FUNCTION_BLOCK jobServiceInterface (* Composite Function Block Type *)
  (* Standard: 61499-2 *)
  (* Version 0.0, 2018-03-05, 4DIAC-IDE, 4DIAC-Consortium *)
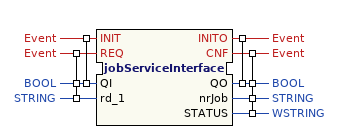
  EVENT_INPUT
    INIT WITH QI; (* Initialization Request *)
    REQ WITH QI, rd_1; (* Normal Execution Request *)
  END_EVENT
  EVENT_OUTPUT
    INITO WITH QO; (* Initialization Confirm *)
    CNF WITH QO, nrJob, STATUS; (* Execution Confirmation *)
  END_EVENT
  VAR_INPUT
    QI : BOOL := TRUE; (* Input event qualifier *)
    rd_1 : STRING;
  END_VAR
  VAR_OUTPUT
    QO : BOOL; (* Output event qualifier *)
    nrJob : STRING;
    STATUS : WSTRING;
  END_VAR
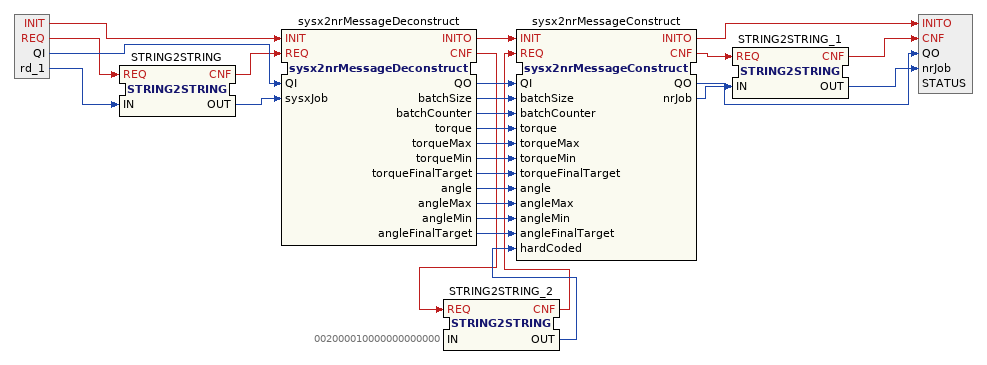
  FBS
    STRING2STRING : STRING2STRING;
    sysx2nrMessageDeconstruct : sysx2nrMessageDeconstruct;
    sysx2nrMessageConstruct : sysx2nrMessageConstruct;
    STRING2STRING_1 : STRING2STRING;
    STRING2STRING_2 : STRING2STRING(IN := 002000010000000000000);
  END_FBS
  EVENT_CONNECTIONS
    STRING2STRING.CNF TO sysx2nrMessageDeconstruct.REQ;
    sysx2nrMessageDeconstruct.INITO TO sysx2nrMessageConstruct.INIT;
    sysx2nrMessageConstruct.INITO TO INITO;
    STRING2STRING_1.CNF TO CNF;
    sysx2nrMessageConstruct.CNF TO STRING2STRING_1.REQ;
    REQ TO STRING2STRING.REQ;
    INIT TO sysx2nrMessageDeconstruct.INIT;
    sysx2nrMessageDeconstruct.CNF TO STRING2STRING_2.REQ;
    STRING2STRING_2.CNF TO sysx2nrMessageConstruct.REQ;
  END_CONNECTIONS
  DATA_CONNECTIONS
    STRING2STRING.OUT TO sysx2nrMessageDeconstruct.sysxJob;
    sysx2nrMessageDeconstruct.QO TO sysx2nrMessageConstruct.QI;
    sysx2nrMessageDeconstruct.batchSize TO sysx2nrMessageConstruct.batchSize;
    sysx2nrMessageDeconstruct.batchCounter TO sysx2nrMessageConstruct.batchCounter;
    sysx2nrMessageDeconstruct.torque TO sysx2nrMessageConstruct.torque;
    sysx2nrMessageDeconstruct.torqueMax TO sysx2nrMessageConstruct.torqueMax;
    sysx2nrMessageDeconstruct.torqueMin TO sysx2nrMessageConstruct.torqueMin;
    sysx2nrMessageDeconstruct.torqueFinalTarget TO sysx2nrMessageConstruct.torqueFinalTarget;
    sysx2nrMessageDeconstruct.angle TO sysx2nrMessageConstruct.angle;
    sysx2nrMessageDeconstruct.angleMax TO sysx2nrMessageConstruct.angleMax;
    sysx2nrMessageDeconstruct.angleMin TO sysx2nrMessageConstruct.angleMin;
    sysx2nrMessageDeconstruct.angleFinalTarget TO sysx2nrMessageConstruct.angleFinalTarget;
    sysx2nrMessageConstruct.QO TO QO;
    sysx2nrMessageConstruct.nrJob TO STRING2STRING_1.IN;
    QI TO sysx2nrMessageDeconstruct.QI;
    rd_1 TO STRING2STRING.IN;
    STRING2STRING_2.OUT TO sysx2nrMessageConstruct.hardCoded;
    STRING2STRING_1.OUT TO nrJob;
  END_CONNECTIONS
END_FUNCTION_BLOCK
